PROGRAM PRG_AtExit01
VAR
	intnFBSensor : FB_Sensors;
	FEdge : F_TRIG;
END_VAR

intnFBSensor (
	iSensor := At_Exit,
	iTimeToActuateSensor := 0,
);

FEdge (
	CLK := intnFBSensor.outSensorON,
	Q => GVL.AtExitPulse,
);

END_PROGRAM

(* stored: Version 1.1.0.1
   POU PRG_AtExit01: Id {864bb69f-ed22-42bd-ad26-22a154b87f8b}, SpecialFunc None *)
